SUBAPPLICATION AUS_AX_SEL_AUS_2_VAL (* Binäre Auswahl für AUS-Werte mit 2 internen initval_AUS und AUS_AX_SEL_AUS. Schaltet per G-Adapter zwischen val0 (G=FALSE) und val1 (G=TRUE) um. *)
  (* Standard: 61499-2; Description: Copyright (c) 2026 Meisterschulen am Ostbahnhof This program and the accompanying materials are made available under the terms of the Eclipse Public License 2.0 which is available at https://www.eclipse.org/legal/epl-2.0/ SPDX-License-Identifier: EPL-2.0 *)
  (* Version 1.0, 2026-09-10, Franz Höpfinger, Meisterschulen am Ostbahnhof, initial implementation *)
  PACKAGE MyLib::sys;
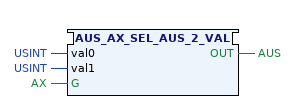
  VAR_INPUT
    val0 : USINT; (* Ausgabewert bei G=FALSE (IN0) *)
    val1 : USINT; (* Ausgabewert bei G=TRUE (IN1) *)
  END_VAR
  SOCKETS
    G : adapter::types::unidirectional::AX; (* Auswahlsignal G *)
  END_SOCKETS
  PLUGS
    OUT : adapter::types::unidirectional::AUS; (* Ausgewaehlter AUS-Adapter Output *)
  END_PLUGS
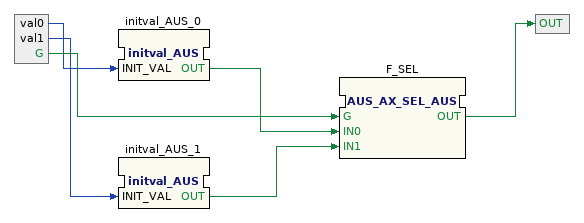
  FBS
    F_SEL : adapter::iec61131::selection::AUS_AX_SEL_AUS;
    initval_AUS_0 : adapter::types::unidirectional::AUS::initval::initval_AUS;
    initval_AUS_1 : adapter::types::unidirectional::AUS::initval::initval_AUS;
  END_FBS
  DATA_CONNECTIONS
    val0 TO initval_AUS_0.INIT_VAL;
    val1 TO initval_AUS_1.INIT_VAL;
  END_CONNECTIONS
  ADAPTER_CONNECTIONS
    G TO F_SEL.G;
    initval_AUS_0.OUT TO F_SEL.IN0;
    initval_AUS_1.OUT TO F_SEL.IN1;
    F_SEL.OUT TO OUT;
  END_CONNECTIONS
END_SUBAPPLICATION
